# EPICS substitutions: hugo/source/db/Beckhoff_4XXX/ecmcEL4732.substitutions
file "ecmcEL47XX-chX.template"
{
  pattern {CH_ID}
          {01   }
          {02   }
}

file "ecmc_analogOutputArray-chX.template"
{
  pattern {CH_ID, DTYP,                FTVL    }
          {01,    "asynInt16ArrayOut", "SHORT" }
          {02,    "asynInt16ArrayOut", "SHORT" }
}

file "ecmcEL37XX_common.template"
{
  pattern {}
          {}
}
